// TIA Portal V17 export
// export: Created 2022-04-06T07:28:41.91165Z, ExportSetting WithDefaults, DisplayName Totally Integrated Automation Portal, DisplayVersion V17, DisplayName TIA Portal Openness, DisplayVersion V17, DisplayName TIA Portal Version Control Interface, DisplayVersion V17, DisplayName TIA Portal Test Suite Advanced, DisplayVersion V17, DisplayName SINAMICS Startdrive Advanced, DisplayVersion V17, DisplayName SINAMICS Startdrive G130, G150, S120, S150, SINAMICS MV, S210, DisplayVersion V17, DisplayName SINAMICS Startdrive G110M, G120, G120C, G120D, G120P, G115D, DisplayVersion V17, DisplayName STEP 7 Professional, DisplayVersion V17, DisplayName STEP 7 Safety, DisplayVersion V17, DisplayName WinCC Advanced / Unified PC, DisplayVersion V17
TYPE "typeFileReadWrite"
// stored: IsFailsafeCompliant false
   STRUCT
      start : Bool;
      offset : UDInt;
      length : UDInt;
      data : Array[0..999] of Byte;
      resultLength : UDInt;
      done : Bool;
      busy : Bool;
      status : Word;
      memErrStatus : Word;
   END_STRUCT;
END_TYPE
